VISUALIZATION V_Option5  // 1160x668
END_VISUALIZATION

(* stored: Version 1.1.0.1, ProductVersion 3.1.4024.3
   Visu V_Option5: Id {c9d53e8f-96cb-4dd0-8bb2-08f03a8d150d} *)
